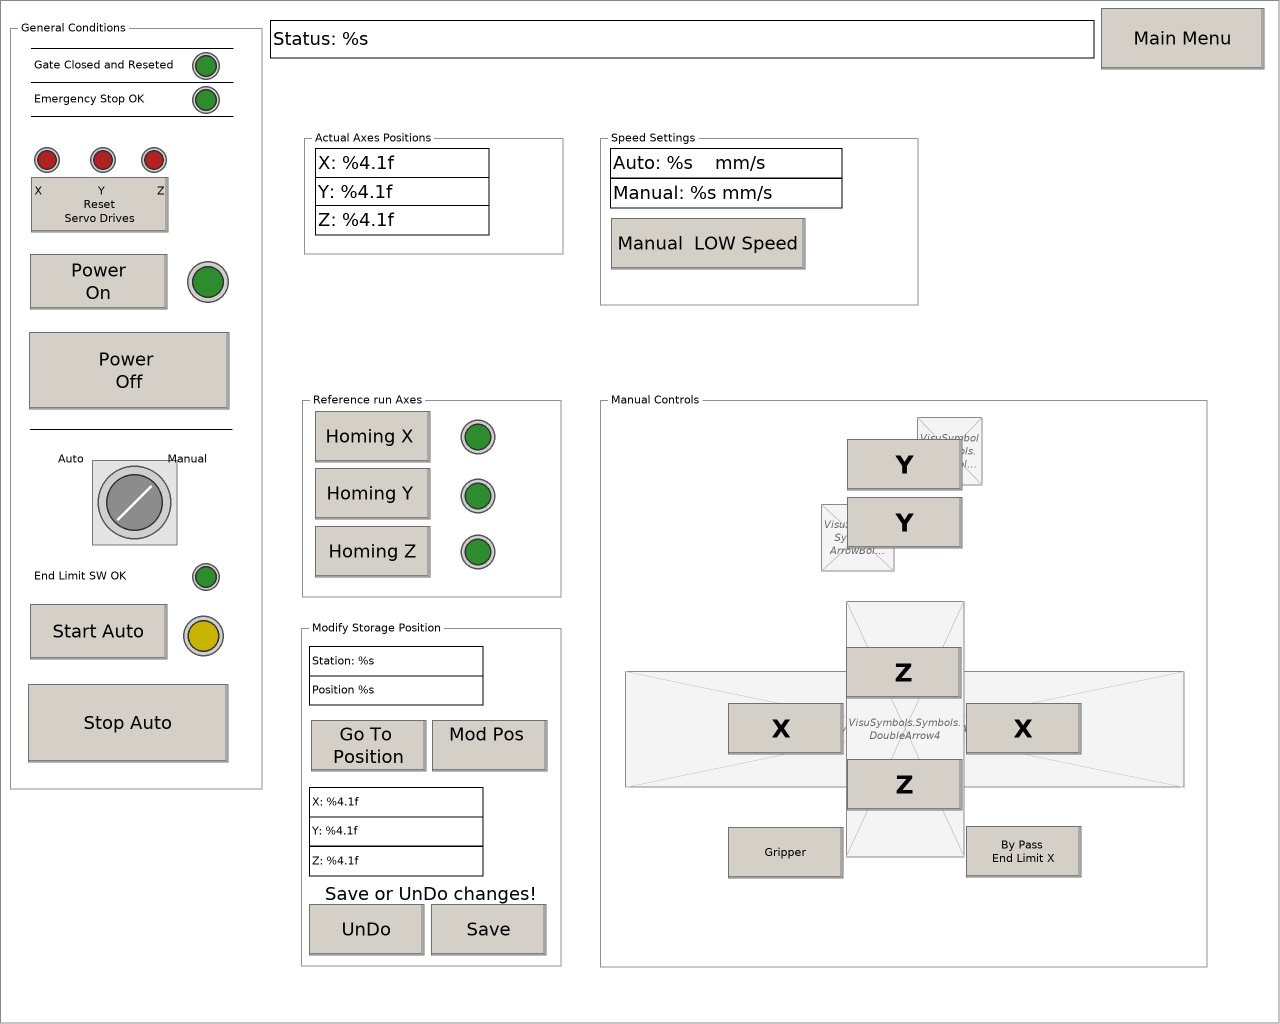
VISUALIZATION GantryRobotVisu  // 1280x1024
    GroupBox (600,392 607x575), "Manual Controls"
        Image (221,112 73x67), image: VisuSymbols.Symbols.ArrowBoldLeftDown
        Image (317,25 65x68), image: VisuSymbols.Symbols.ArrowBoldRightUp
        Image (25,279 559x116), image: VisuSymbols.Symbols.DoubleArrow3
        Image (246,209 118x256), image: VisuSymbols.Symbols.DoubleArrow4
        Button (247,105 115x51), "Y", input disabled if: NOT GantryRobotMotion.mxManualMode
            tap GantryRobotMotion.mxMCYButtonJogFWD
        Button (247,47 115x51), "Y", input disabled if: NOT GantryRobotMotion.mxManualMode
            tap GantryRobotMotion.mxMCYButtonJogBWD
        Button (128,435 115x51), "Gripper", input disabled if: NOT GantryRobotMotion.mxManualMode
            tap GantryRobotMotion.mxTogleGripper
        Button (366,434 115x51), "By Pass End Limit X", invisible if: NOT GantryRobotMotion.mxManualMode, input disabled if: NOT GVL.ixLimSwX
            toggle GantryRobotMotion.mxMCXButtonByPass
        Button (247,367 115x51), "Z", input disabled if: NOT GantryRobotMotion.mxManualMode
            tap GantryRobotMotion.mxMCZButtonJogFWD
        Button (246,255 115x51), "Z", input disabled if: NOT GantryRobotMotion.mxManualMode
            tap GantryRobotMotion.mxMCZButtonJogBWD
        Button (366,311 115x51), "X", input disabled if: NOT GantryRobotMotion.mxManualMode
            tap GantryRobotMotion.mxMCXButtonJogBWD
        Button (128,311 115x51), "X", input disabled if: NOT GantryRobotMotion.mxManualMode
            tap GantryRobotMotion.mxMCXButtonJogFWD
    GroupBox (10,20 252x769), "General Conditions"
        Button (20,234 137x55), "Power On", input disabled if: NOT GantryRobotMotion.mxGeneralCOntrolOk
            tap GantryRobotMotion.mxButtonGeneralControlOn
        Label (21,36 150x32)
        Label (21,29 160x32), "Gate Closed and Reseted"
        Lamp1 (178,30 36x32), variable: GVL.ixLightBeamAndGatesClosed, style: Lamp-Lamp1-Green
        Label (21,63 157x32), "Emergency Stop OK"
        Lamp1 (178,64 36x32), variable: GVL.ixEmergencyStopOk, style: Lamp-Lamp1-Green
        Lamp1 (170,238 56x48), variable: GVL.qxIndControlOn, style: Lamp-Lamp1-Green
        Lamp1 (170,592 47x48), variable: GVL.qxIndProgramStart, style: Lamp-Lamp1-Yellow
        Label (21,540 120x32), "End Limit SW OK"
        Lamp1 (178,541 36x32), variable: GantryRobotMotion.mxLimSwOK, style: Lamp-Lamp1-Green
        Line (21,28) (223,28)
        Line (21,62) (223,62)
        Line (21,96) (223,96)
        RotarySwitch (75,440 99x85), variable: GantryRobotMotion.mxButtonAutoMode, behaviour: TOGGLE, style: Switch-RotarySwitch-Gray
        Label (26,423 193x32), "Auto Manual"
        Line (20,409) (222,409)
        Button (20,584 137x55), "Start Auto", input disabled if: NOT GantryRobotMotion.mxAutoMode
            tap GantryRobotMotion.mxButtonStartAuto
        Lamp1 (128,125 32x30), variable: GantryRobotMotion.mxMCXAxisError, style: Lamp-Lamp1-Red
        Lamp1 (77,125 32x30), variable: GantryRobotMotion.mxMCXAxisError, style: Lamp-Lamp1-Red
        Lamp1 (21,125 32x30), variable: GantryRobotMotion.mxMCXAxisError, style: Lamp-Lamp1-Red
        Button (21,157 137x55), "X Y Z Reset Servo Drives"
            tap GantryRobotMotion.mxButtonResetError
        Button (19,312 200x77), "Power Off", input disabled if: NOT GantryRobotMotion.mxGeneralCOntrolOk
            tap GantryRobotMotion.mxButtonGeneralControlOff
        Button (18,664 200x78), "Stop Auto", input disabled if: NOT GantryRobotMotion.mxAutoMode
            tap GantryRobotMotion.mxButtonStopAuto
    GroupBox (304,130 259x124), "Actual Axes Positions"
        Rectangle (11,18 174x30), "X: %4.1f", text variable: GantryRobotMotion.MCActualPos.x
        Rectangle (11,47 174x30), "Y: %4.1f", text variable: GantryRobotMotion.MCActualPos.y
        Rectangle (11,75 174x30), "Z: %4.1f", text variable: GantryRobotMotion.MCActualPos.z
    Button (1101,8 163x61), "Main Menu"
        OnMouseClick: change screen: Visualization
    Rectangle (270,20 824x38), "Status: %s", text variable: GantryRobotMotion.strStatusText
    GroupBox (600,130 318x175), "Speed Settings"
        Rectangle (10,18 232x30), "Auto: %s mm/s", text variable: GantryRobotMotion.MCAutoVelocity
            OnMouseClick: write the text variable via VisuDialogs.Numpad, min 100, max 1000, title 'Auto Speed mm/s', format %i
        Rectangle (10,48 232x30), "Manual: %s mm/s", text variable: GantryRobotMotion.MCJogVelocity
            OnMouseClick: write the text variable via VisuDialogs.Numpad, min 5, max 250, title 'Jog Speed mm/s', format %i
        Button (11,88 194x51), "Manual LOW Speed", input disabled if: NOT GantryRobotMotion.mxManualMode
            toggle GantryRobotMotion.mxMCButtonManLowVelocity
    GroupBox (301,620 260x346), "Modify Storage Position"
        Button (131,100 115x51), "Mod Pos", input disabled if: NOT GantryRobotMotion.mxManualMode OR NOT GantryRobotMotion.mxHomingDone
            tap GantryRobotMotion.mxButtonModPosExecute
        Rectangle (8,55 174x30), "Position %s", text variable: GantryRobotMotion.ModPosLocation, input disabled if: NOT GantryRobotMotion.mxManualMode
            OnMouseClick: write GantryRobotMotion.ModPosLocation via VisuDialogs.Numpad, min 1, max 9, title "Loacation", format %i
        Button (10,100 115x51), "Go To Position", input disabled if: NOT GantryRobotMotion.mxManualMode OR NOT GantryRobotMotion.mxHomingDone
            tap GantryRobotMotion.mxButtonGoToModPos
        Rectangle (8,26 174x30), "Station: %s", text variable: GantryRobotMotion.ModPosStation, input disabled if: NOT GantryRobotMotion.mxManualMode
            OnMouseClick: write GantryRobotMotion.ModPosStation via VisuDialogs.Numpad, min 1, max 4, title "Station", format %i
        Rectangle (8,196 174x30), "Y: %4.1f", text variable: GantryRobotMotion.arrAbsPosition[GantryRobotMotion.ModPosStation, GantryRobotMotion.ModPosLocation].y, input disabled if: NOT GantryRobotMotion.mxManualMode
            OnMouseClick: write the text variable via VisuDialogs.Numpad, title 'Position Y', format %f
            OnMouseClick: execute { GantryRobotMotion.mxReminderToSave := TRUE; }
        Rectangle (8,226 174x30), "Z: %4.1f", text variable: GantryRobotMotion.arrAbsPosition[GantryRobotMotion.ModPosStation, GantryRobotMotion.ModPosLocation].z, input disabled if: NOT GantryRobotMotion.mxManualMode
            OnMouseClick: write the text variable via VisuDialogs.Numpad, title 'Position Z', format %f
            OnMouseClick: execute { GantryRobotMotion.mxReminderToSave := TRUE; }
        Button (130,284 115x51), "Save", input disabled if: NOT GantryRobotMotion.mxManualMode
            tap GantryRobotMotion.mxButtonSavePos
        Button (8,284 115x51), "UnDo", input disabled if: NOT GantryRobotMotion.mxManualMode
            tap GantryRobotMotion.mxButtonReadFile
        Rectangle (8,167 174x30), "X: %4.1f", text variable: GantryRobotMotion.arrAbsPosition[GantryRobotMotion.ModPosStation, GantryRobotMotion.ModPosLocation].x, input disabled if: NOT GantryRobotMotion.mxManualMode
            OnMouseClick: write the text variable via VisuDialogs.Numpad, title 'Position Z', format %f
            OnMouseClick: execute { GantryRobotMotion.mxReminderToSave := TRUE; }
    GroupBox (302,392 259x205), "Reference run Axes"
        Lamp1 (156,140 40x40), variable: GantryRobotMotion.mxMCZHomingDone, style: Lamp-Lamp1-Green
        Lamp1 (156,84 40x40), variable: GantryRobotMotion.mxMCYHomingDone, style: Lamp-Lamp1-Green
        Lamp1 (156,25 40x40), variable: GantryRobotMotion.mxMCXHomingDone, style: Lamp-Lamp1-Green
        Button (13,134 115x51), "Homing Z", input disabled if: NOT GantryRobotMotion.mxManualMode
            tap GantryRobotMotion.mxMCZButtonHoming
        Button (13,76 115x51), "Homing Y", input disabled if: NOT GantryRobotMotion.mxManualMode
            tap GantryRobotMotion.mxMCYButtonHoming
        Button (13,19 115x51), "Homing X", input disabled if: NOT GantryRobotMotion.mxManualMode
            tap GantryRobotMotion.mxMCXButtonHoming
    Label (306,880 250x28), "Save or UnDo changes!", invisible if: NOT GantryRobotMotion.mxReminderToSave
END_VISUALIZATION

(* stored: Version 1.1.0.1, ProductVersion 3.1.4022.12
   Visu GantryRobotVisu: Id {00b2fabf-60ad-4184-b41c-b3b945dff1fc} *)
